FUNCTION Convert_DT_TO_USINT : Hresult
VAR_INPUT
	in : DT;
	out : REFERENCE TO USINT;
END_VAR
VAR
	converted : USINT;
END_VAR

converted := DT_TO_USINT(in);

IF (USINT_TO_DT(converted) <> in) THEN
	Convert_DT_TO_USINT := INCOMPATIBLE;
	RETURN;
END_IF

out := converted;

END_FUNCTION

(* stored: Version 1.1.0.1, ProductVersion 3.1.4024.12
   POU Convert_DT_TO_USINT: Id {fb92529c-5682-49ef-9223-5835f533d533}, SpecialFunc None *)
